FUNCTION_BLOCK FB_ESSMonitoringMCU500x
VAR_INPUT
    nEcMasterNetId: T_AmsNetId;
END_VAR
VAR_OUTPUT
    aErrorID: ARRAY [1..nMaxAlarms] OF INT;
    aErrorMsg: ARRAY [1..nMaxAlarms] OF STRING;
    nEcMasterFramesLost: UDINT;
    nCPULoad: UDINT;
    fCycleExecTime_ms: REAL;
    nAlarmGrpBitNumber: UDINT;
END_VAR
VAR
    //Outputs
    {attribute 'TcLinkTo' := 'TIID^Device 2 (EtherCAT)^Term 1 (EK1100)^Term 8 (EL2014)^DIG Outputs^Channel 1^Output'}
    bStatusLED AT %Q*: BOOL;
    {attribute 'TcLinkTo' := 'TIID^Device 2 (EtherCAT)^Term 1 (EK1100)^Term 7 (EL2014)^DIG Outputs^Channel 4^Output'}
    bAcknowledgeLED AT %Q*: BOOL;
    {attribute 'TcLinkTo' := 'TIID^Device 2 (EtherCAT)^Term 1 (EK1100)^Term 8 (EL2014)^DIG Outputs^Channel 2^Output'}
    bEStopLED AT %Q*: BOOL;
    {attribute 'TcLinkTo' := 'TIID^Device 2 (EtherCAT)^Term 1 (EK1100)^Term 8 (EL2014)^DIG Outputs^Channel 3^Output'}
    bEmergencyLED AT %Q*: BOOL;
    {attribute 'TcLinkTo' := 'TIID^Device 2 (EtherCAT)^Term 1 (EK1100)^Term 8 (EL2014)^DIG Outputs^Channel 4^Output'}
    bAbnormalLED AT %Q*: BOOL;

    //Inputs
    {attribute 'TcLinkTo' := 'TIID^Device 2 (EtherCAT)^Term 1 (EK1100)^Term 4 (EL1808)^Channel 1^Input'}
    b24VDC1_OK AT %I*: BOOL;
    {attribute 'TcLinkTo' := 'TIID^Device 2 (EtherCAT)^Term 1 (EK1100)^Term 4 (EL1808)^Channel 2^Input'}
    b24VDC2_OK AT %I*: BOOL;
    {attribute 'TcLinkTo' := 'TIID^Device 2 (EtherCAT)^Term 1 (EK1100)^Term 4 (EL1808)^Channel 3^Input'}
    b24VDC3_OK AT %I*: BOOL;
    {attribute 'TcLinkTo' := 'TIID^Device 2 (EtherCAT)^Term 1 (EK1100)^Term 4 (EL1808)^Channel 4^Input'}
    b48VDC1_OK AT %I*: BOOL;
    {attribute 'TcLinkTo' := 'TIID^Device 2 (EtherCAT)^Term 1 (EK1100)^Term 4 (EL1808)^Channel 5^Input'}
    b48VDC2_OK AT %I*: BOOL;
    {attribute 'TcLinkTo' := 'TIID^Device 2 (EtherCAT)^Term 1 (EK1100)^Term 4 (EL1808)^Channel 6^Input'}
    b48VDC3_OK AT %I*: BOOL;
    {attribute 'TcLinkTo' := 'TIID^Device 2 (EtherCAT)^Term 1 (EK1100)^Term 4 (EL1808)^Channel 7^Input'}
    b48VDC4_OK AT %I*: BOOL;
    {attribute 'TcLinkTo' := 'TIID^Device 2 (EtherCAT)^Term 1 (EK1100)^Term 3 (EL1808)^Channel 1^Input'}
    bFuse1_OK AT %I*: BOOL;
    {attribute 'TcLinkTo' := 'TIID^Device 2 (EtherCAT)^Term 1 (EK1100)^Term 3 (EL1808)^Channel 2^Input'}
    bFuse2_OK AT %I*: BOOL;
    {attribute 'TcLinkTo' := 'TIID^Device 2 (EtherCAT)^Term 1 (EK1100)^Term 3 (EL1808)^Channel 3^Input'}
    bFuse3_OK AT %I*: BOOL;
    {attribute 'TcLinkTo' := 'TIID^Device 2 (EtherCAT)^Term 1 (EK1100)^Term 3 (EL1808)^Channel 4^Input'}
    bFuse4_OK AT %I*: BOOL;
    {attribute 'TcLinkTo' := 'TIID^Device 2 (EtherCAT)^Term 1 (EK1100)^Term 3 (EL1808)^Channel 5^Input'}
    bFuse5_OK AT %I*: BOOL;
    {attribute 'TcLinkTo' := 'TIID^Device 2 (EtherCAT)^Term 1 (EK1100)^Term 3 (EL1808)^Channel 6^Input'}
    bFuse6_OK AT %I*: BOOL;
    {attribute 'TcLinkTo' := 'TIID^Device 2 (EtherCAT)^Term 1 (EK1100)^Term 3 (EL1808)^Channel 7^Input'}
    bFuse7_OK AT %I*: BOOL;
    {attribute 'TcLinkTo' := 'TIID^Device 2 (EtherCAT)^Term 1 (EK1100)^Term 3 (EL1808)^Channel 8^Input'}
    bFuse8_OK AT %I*: BOOL;
    {attribute 'TcLinkTo' := 'TIID^Device 2 (EtherCAT)^Term 1 (EK1100)^Term 5 (EL1808)^Channel 1^Input'}
    bEStop1Triggered AT %I*: BOOL;
    {attribute 'TcLinkTo' := 'TIID^Device 2 (EtherCAT)^Term 1 (EK1100)^Term 5 (EL1808)^Channel 2^Input'}
    bSTO1Triggered AT %I*: BOOL;
    {attribute 'TcLinkTo' := 'TIID^Device 2 (EtherCAT)^Term 1 (EK1100)^Term 5 (EL1808)^Channel 3^Input'}
    bEStop2Triggered AT %I*: BOOL;
    {attribute 'TcLinkTo' := 'TIID^Device 2 (EtherCAT)^Term 1 (EK1100)^Term 5 (EL1808)^Channel 4^Input'}
    bSTO2Triggered AT %I*: BOOL;
    {attribute 'TcLinkTo' := 'TIID^Device 2 (EtherCAT)^Term 1 (EK1100)^Term 6 (EL1808)^Channel 2^Input'}
    bMCB_OK AT %I*: BOOL;
    {attribute 'TcLinkTo' := 'TIID^Device 2 (EtherCAT)^Term 1 (EK1100)^Term 6 (EL1808)^Channel 3^Input'}
    bSPD_OK AT %I*: BOOL;
    {attribute 'TcLinkTo' := 'TIID^Device 2 (EtherCAT)^Term 1 (EK1100)^Term 6 (EL1808)^Channel 4^Input'}
    bDoorClosed AT %I*: BOOL;
    {attribute 'TcLinkTo' := 'TIID^Device 2 (EtherCAT)^Term 1 (EK1100)^Term 6 (EL1808)^Channel 5^Input'}
    bAcknowledgeButton AT %I*: BOOL;
    {attribute 'TcLinkTo' := 'TIID^Device 2 (EtherCAT)^Term 1 (EK1100)^Term 9 (EL3214)^RTD Inputs Channel 1^Value'}
    nTemp1 AT %I*: INT;
    {attribute 'TcLinkTo' := 'TIID^Device 2 (EtherCAT)^Term 1 (EK1100)^Term 9 (EL3214)^RTD Inputs Channel 2^Value'}
    nTemp2 AT %I*: INT;
    {attribute 'TcLinkTo' := 'TIID^Device 2 (EtherCAT)^Term 1 (EK1100)^Term 9 (EL3214)^RTD Inputs Channel 3^Value'}
    nTemp3 AT %I*: INT;
    {attribute 'TcLinkTo' := 'TIID^Device 2 (EtherCAT)^Term 1 (EK1100)^Term 9 (EL3214)^RTD Inputs Channel 4^Value'}
    nTemp4 AT %I*: INT;
    {attribute 'TcLinkTo' := 'TIID^Device 2 (EtherCAT)^Inputs^DevState'}
    nEcMasterDevState AT %I*: UINT;

    aAlarmList: ARRAY [1..nMaxAlarms] OF ST_MonitoringAlarm := [
(*[1]*)(nErrorID:=241, sErrorMsg:='The DC OK Status from PS 24V-1 is OFF.', nStatusLED:=E_MonitoringLedFunction.eFast, nAbnormalLED:=E_MonitoringLedFunction.eSteady, nEmergencyLED:=E_MonitoringLedFunction.eSteady, nAcknowledgeLED:=E_MonitoringLedFunction.eSteady),
(*[2]*)(nErrorID:=242, sErrorMsg:='The DC OK Status from PS 24V-2 is OFF.', nStatusLED:=E_MonitoringLedFunction.eFast, nAbnormalLED:=E_MonitoringLedFunction.eSteady, nEmergencyLED:=E_MonitoringLedFunction.eSteady, nAcknowledgeLED:=E_MonitoringLedFunction.eSteady),
(*[3]*)(nErrorID:=243, sErrorMsg:='The DC OK Status from PS 24V-3 is OFF.', nStatusLED:=E_MonitoringLedFunction.eFast, nAbnormalLED:=E_MonitoringLedFunction.eSteady, nEmergencyLED:=E_MonitoringLedFunction.eSteady, nAcknowledgeLED:=E_MonitoringLedFunction.eSteady),
(*[4]*)(nErrorID:=481, sErrorMsg:='The DC OK Status from PS 48V-1 is OFF.', nStatusLED:=E_MonitoringLedFunction.eFast, nAbnormalLED:=E_MonitoringLedFunction.eSteady, nEmergencyLED:=E_MonitoringLedFunction.eSteady, nAcknowledgeLED:=E_MonitoringLedFunction.eSteady),
(*[5]*)(nErrorID:=482, sErrorMsg:='The DC OK Status from PS 48V-2 is OFF.', nStatusLED:=E_MonitoringLedFunction.eFast, nAbnormalLED:=E_MonitoringLedFunction.eSteady, nEmergencyLED:=E_MonitoringLedFunction.eSteady, nAcknowledgeLED:=E_MonitoringLedFunction.eSteady),
(*[6]*)(nErrorID:=483, sErrorMsg:='The DC OK Status from PS 48V-3 is OFF.', nStatusLED:=E_MonitoringLedFunction.eFast, nAbnormalLED:=E_MonitoringLedFunction.eSteady, nEmergencyLED:=E_MonitoringLedFunction.eSteady, nAcknowledgeLED:=E_MonitoringLedFunction.eSteady),
(*[7]*)(nErrorID:=484, sErrorMsg:='The DC OK Status from PS 48V-4 is OFF.', nStatusLED:=E_MonitoringLedFunction.eFast, nAbnormalLED:=E_MonitoringLedFunction.eSteady, nEmergencyLED:=E_MonitoringLedFunction.eSteady, nAcknowledgeLED:=E_MonitoringLedFunction.eSteady),
(*[8]*)(nErrorID:=11, sErrorMsg:='MCB OK status is OFF', nStatusLED:=E_MonitoringLedFunction.eFast, nAbnormalLED:=E_MonitoringLedFunction.eSteady, nEmergencyLED:=E_MonitoringLedFunction.eSteady, nAcknowledgeLED:=E_MonitoringLedFunction.eSteady),
(*[9]*)(nErrorID:=12, sErrorMsg:='SPD OK status is OFF', nStatusLED:=E_MonitoringLedFunction.eFast, nAbnormalLED:=E_MonitoringLedFunction.eSteady, nEmergencyLED:=E_MonitoringLedFunction.eSteady, nAcknowledgeLED:=E_MonitoringLedFunction.eSteady),
(*[10]*)(nErrorID:=13, sErrorMsg:='Cabinet door Opened', nStatusLED:=E_MonitoringLedFunction.eSteady, nAbnormalLED:=E_MonitoringLedFunction.eSteady, nEmergencyLED:=E_MonitoringLedFunction.eSteady, nAcknowledgeLED:=E_MonitoringLedFunction.eUndefined),
(*[11]*)(nErrorID:=301, sErrorMsg:='Fuse 1 tripped', nStatusLED:=E_MonitoringLedFunction.eUndefined, nAbnormalLED:=E_MonitoringLedFunction.eSteady, nEmergencyLED:=E_MonitoringLedFunction.eUndefined, nAcknowledgeLED:=E_MonitoringLedFunction.eSteady),
(*[12]*)(nErrorID:=302, sErrorMsg:='Fuse 2 tripped', nStatusLED:=E_MonitoringLedFunction.eSlow, nAbnormalLED:=E_MonitoringLedFunction.eSteady, nEmergencyLED:=E_MonitoringLedFunction.eSteady, nAcknowledgeLED:=E_MonitoringLedFunction.eSteady),
(*[13]*)(nErrorID:=303, sErrorMsg:='Fuse 3 tripped', nStatusLED:=E_MonitoringLedFunction.eSlow, nAbnormalLED:=E_MonitoringLedFunction.eSteady, nEmergencyLED:=E_MonitoringLedFunction.eSteady, nAcknowledgeLED:=E_MonitoringLedFunction.eSteady),
(*[14]*)(nErrorID:=304, sErrorMsg:='Fuse 4 tripped', nStatusLED:=E_MonitoringLedFunction.eSlow, nAbnormalLED:=E_MonitoringLedFunction.eSteady, nEmergencyLED:=E_MonitoringLedFunction.eUndefined, nAcknowledgeLED:=E_MonitoringLedFunction.eSteady),
(*[15]*)(nErrorID:=305, sErrorMsg:='Fuse 5 tripped', nStatusLED:=E_MonitoringLedFunction.eSlow, nAbnormalLED:=E_MonitoringLedFunction.eSteady, nEmergencyLED:=E_MonitoringLedFunction.eUndefined, nAcknowledgeLED:=E_MonitoringLedFunction.eSteady),
(*[16]*)(nErrorID:=306, sErrorMsg:='Fuse 6 tripped', nStatusLED:=E_MonitoringLedFunction.eSlow, nAbnormalLED:=E_MonitoringLedFunction.eSteady, nEmergencyLED:=E_MonitoringLedFunction.eUndefined, nAcknowledgeLED:=E_MonitoringLedFunction.eSteady),
(*[17]*)(nErrorID:=307, sErrorMsg:='Fuse 7 tripped', nStatusLED:=E_MonitoringLedFunction.eSlow, nAbnormalLED:=E_MonitoringLedFunction.eSteady, nEmergencyLED:=E_MonitoringLedFunction.eUndefined, nAcknowledgeLED:=E_MonitoringLedFunction.eSteady),
(*[18]*)(nErrorID:=308, sErrorMsg:='Fuse 8 tripped', nStatusLED:=E_MonitoringLedFunction.eSlow, nAbnormalLED:=E_MonitoringLedFunction.eSteady, nEmergencyLED:=E_MonitoringLedFunction.eUndefined, nAcknowledgeLED:=E_MonitoringLedFunction.eSteady),
(*[19]*)(nErrorID:=501, sErrorMsg:='E-Stop 1 active', nStatusLED:=E_MonitoringLedFunction.eSteady, nAbnormalLED:=E_MonitoringLedFunction.eSteady, nEmergencyLED:=E_MonitoringLedFunction.eUndefined, nAcknowledgeLED:=E_MonitoringLedFunction.eUndefined, nEStopLED:=E_MonitoringLedFunction.eSteady),
(*[20]*)(nErrorID:=511, sErrorMsg:='STO axis 1 active', nStatusLED:=E_MonitoringLedFunction.eFast, nAbnormalLED:=E_MonitoringLedFunction.eSteady, nEmergencyLED:=E_MonitoringLedFunction.eUndefined, nAcknowledgeLED:=E_MonitoringLedFunction.eUndefined),
(*[21]*)(nErrorID:=502, sErrorMsg:='E-Stop 2 active', nStatusLED:=E_MonitoringLedFunction.eSteady, nAbnormalLED:=E_MonitoringLedFunction.eSteady, nEmergencyLED:=E_MonitoringLedFunction.eUndefined, nAcknowledgeLED:=E_MonitoringLedFunction.eUndefined, nEStopLED:=E_MonitoringLedFunction.eSteady),
(*[22]*)(nErrorID:=512, sErrorMsg:='STO axis 2 active', nStatusLED:=E_MonitoringLedFunction.eFast, nAbnormalLED:=E_MonitoringLedFunction.eSteady, nEmergencyLED:=E_MonitoringLedFunction.eUndefined, nAcknowledgeLED:=E_MonitoringLedFunction.eUndefined),
(*[23]*)(nErrorID:=14, sErrorMsg:='Temperature 1 too high', nStatusLED:=E_MonitoringLedFunction.eUndefined, nAbnormalLED:=E_MonitoringLedFunction.eSteady, nEmergencyLED:=E_MonitoringLedFunction.eSteady, nAcknowledgeLED:=E_MonitoringLedFunction.eUndefined),
(*[24]*)(nErrorID:=15, sErrorMsg:='Temperature 2 too high', nStatusLED:=E_MonitoringLedFunction.eUndefined, nAbnormalLED:=E_MonitoringLedFunction.eSteady, nEmergencyLED:=E_MonitoringLedFunction.eSteady, nAcknowledgeLED:=E_MonitoringLedFunction.eUndefined),
(*[25]*)(nErrorID:=16, sErrorMsg:='Temperature 3 too high', nStatusLED:=E_MonitoringLedFunction.eUndefined, nAbnormalLED:=E_MonitoringLedFunction.eSteady, nEmergencyLED:=E_MonitoringLedFunction.eSteady, nAcknowledgeLED:=E_MonitoringLedFunction.eUndefined),
(*[26]*)(nErrorID:=17, sErrorMsg:='Temperature 4 too high', nStatusLED:=E_MonitoringLedFunction.eUndefined, nAbnormalLED:=E_MonitoringLedFunction.eSteady, nEmergencyLED:=E_MonitoringLedFunction.eSteady, nAcknowledgeLED:=E_MonitoringLedFunction.eUndefined),
(*[27]*)(nErrorID:=101, sErrorMsg:='EtherCAT Master is not ok', nStatusLED:=E_MonitoringLedFunction.eSteady, nAbnormalLED:=E_MonitoringLedFunction.eSlow, nEmergencyLED:=E_MonitoringLedFunction.eUndefined, nAcknowledgeLED:=E_MonitoringLedFunction.eUndefined),
(*[28]*)(nErrorID:=102, sErrorMsg:='At least one EtherCAT slave is not in OP state', nStatusLED:=E_MonitoringLedFunction.eSteady, nAbnormalLED:=E_MonitoringLedFunction.eSlow, nEmergencyLED:=E_MonitoringLedFunction.eSteady, nAcknowledgeLED:=E_MonitoringLedFunction.eUndefined),
(*[29]*)(nErrorID:=103, sErrorMsg:='At least one EtherCAT slave link is faulted', nStatusLED:=E_MonitoringLedFunction.eSteady, nAbnormalLED:=E_MonitoringLedFunction.eSlow, nEmergencyLED:=E_MonitoringLedFunction.eSteady, nAcknowledgeLED:=E_MonitoringLedFunction.eUndefined),
(*[30]*)(nErrorID:=104, sErrorMsg:='Overflow in PLC cycle time', nStatusLED:=E_MonitoringLedFunction.eSteady, nAbnormalLED:=E_MonitoringLedFunction.eSlow, nEmergencyLED:=E_MonitoringLedFunction.eUndefined, nAcknowledgeLED:=E_MonitoringLedFunction.eUndefined),
(*[31]*)(nErrorID:=105, sErrorMsg:='CPU Load High', nStatusLED:=E_MonitoringLedFunction.eSteady, nAbnormalLED:=E_MonitoringLedFunction.eSlow, nEmergencyLED:=E_MonitoringLedFunction.eUndefined, nAcknowledgeLED:=E_MonitoringLedFunction.eUndefined)];

    aTempErrorID: ARRAY [1..nMaxAlarms] OF INT;
    aTempErrorMsg: ARRAY [1..nMaxAlarms] OF STRING;

    aFbErrorMessageTimer: ARRAY[1..nMaxAlarms] OF TON;
    aStartErrorMsgTimer: ARRAY[1..nMaxAlarms] OF BOOL;
    aFbErrorTrig: ARRAY[1..nMaxAlarms] OF R_TRIG;

    nLEDAlarmID: INT;
    nAlarmCnt: INT;
    nAlarmBitNumber: UDINT;

    bCPUOverloaded: BOOL;
    bEcMasterError: BOOL;
    bSlaveStateNotOP: BOOL;
    bSlaveLinkError: BOOL;
    aExtraMessage: ARRAY[1..nMaxAlarms] OF STRING := [nMaxAlarms('')];
    bCycleTimeExceeded: BOOL;
    //Cpu Monitor
    fbMonitorCPU: TC_CpuUsage;
    fbUpdateCPULoadTON: TON;
    fMaxCPULoad: USINT := 85;
    //Ethercat master device state
    bEcLinkError: BOOL;
    bEcIOlocked: BOOL;
    bEcLinkErrorRedundancyAdapter: BOOL;
    bEcMissingFrame: BOOL;
    bEcOutofSendResources: BOOL;
    bEcWatchdogTriggered: BOOL;
    bEcEthernetDriverNotFound: BOOL;
    bEcIOresetActive: BOOL;
    bEcSlaveINIT: BOOL;
    bEcSlavePreOP: BOOL;
    bEcSlaveSafeOP: BOOL;
    bEcSlaveError: BOOL;
    bEcDCnotInSync: BOOL;
    //Ehtercat slave device state
    fbUpdateEcSlaveStateTON: TON;
    fbGetEcSlaveStates: FB_EcGetAllSlaveStates;
    stSlaveState: ARRAY[0..nMaxECSlaves] OF ST_EcSlaveState;
    nActualEcSlaves: INT := 0;
    i: INT;
    //Frame statistics
    fbUpdateEcMasterFrame: TON;
    fbGetEcMasterFrames: FB_EcMasterFrameStatistic;

    nAcknowledgeLED: E_MonitoringLedFunction;
    nStatusLED: E_MonitoringLedFunction;
    nAbnormalLED: E_MonitoringLedFunction;
    nEmergencyLED: E_MonitoringLedFunction;
    fbFastBlinkOn: TON;
    fbFastBlinkOff: TON;
    bFastBlink: BOOL;
    fbSlowBlinkOn: TON;
    fbSlowBlinkOff: TON;
    bSlowBlink: BOOL;

    fbAcknowledgeButtonTrig: R_TRIG;

    fbEtherCATAlarmDelayTON: TON;
    bStartEtherCATdelayTON: BOOL := FALSE;
    bEtherCATInitialized: BOOL := FALSE;
END_VAR
VAR CONSTANT
    nMaxAlarms: INT := 50;
    nMaxECSlaves: INT := 255;
    nMaxTemp: INT := 10000;
    nSlaveStateNotOPEntry: UDINT := 28;
    nSlaveLinkErrorEntry: UDINT := 29;
END_VAR

actMonitorAlarms();
actMonitorCPU();
actMonitorEtherCAT();

ACTION actMonitorAlarms:
fbAcknowledgeButtonTrig(CLK:=bAcknowledgeButton);
mSetResetAlarmsLeds();

// Reset before loop
nAlarmCnt := 0;
nAlarmBitNumber := 0;
MEMSET(ADR(aTempErrorID), 0, SIZEOF(aTempErrorID));
MEMSET(ADR(aTempErrorMsg), 0, SIZEOF(aTempErrorMsg));
nLEDAlarmID := 0;
nEmergencyLED := 0;
nAbnormalLED := 0;
nStatusLED := 0;
nAcknowledgeLED := 0;

FOR i:=1 TO nMaxAlarms DO
    afbErrorMessageTimer[i](IN:=aStartErrorMsgTimer[i], PT:=T#60S);
    aFbErrorTrig[i](clk:=aStartErrorMsgTimer[i]);
    // Update list of active alarms
    mAlarm(stAlarmData:=aAlarmList[i]);
    // Update list of active LEDs
    mLed(stAlarmData:=aAlarmList[i]);

    IF aAlarmList[i].bAlarmActive THEN
        nAlarmCnt := nAlarmCnt + 1;
        aTempErrorID[nAlarmCnt] := aAlarmList[i].nErrorID;
        aTempErrorMsg[nAlarmCnt] := CONCAT(aAlarmList[i].sErrorMsg, aExtraMessage[i]);

        mPrintErrorMessage(
            sErrorMessage:=aTempErrorMsg[nAlarmCnt],
            nErrorID:=aAlarmList[i].nErrorID);

        // Map nErrorID to nAlarmBitnumber, which later is mapped to output variable nAlarmGrpBitNumber.
        CASE aAlarmList[i].nErrorID OF
            1,4:
            nAlarmBitNumber.0 := TRUE;
            9,12,13:
            nAlarmBitNumber.1 := TRUE;
            10,11:
            nAlarmBitNumber.2 := TRUE;
            14,15:
            nAlarmBitNumber.3 := TRUE;
            21,22:
            nAlarmBitNumber.4 := TRUE;
            23,24:
            nAlarmBitNumber.5 := TRUE;
            104,105:
            nAlarmBitNumber.6 := TRUE;
            103:
            nAlarmBitNumber.7 := TRUE;
            102:
            nAlarmBitNumber.8 := TRUE;
            30:
            nAlarmBitNumber.9 := TRUE;
        END_CASE
    END_IF

    // Set the alarm LEDs according to first occurrence
    IF nLEDAlarmID = 0 AND aALarmList[i].bLedActive THEN
        nLEDAlarmID := i;
        nEmergencyLED := aAlarmList[i].nEmergencyLED;
        nAbnormalLED := aAlarmList[i].nAbnormalLED;
        nStatusLED := aAlarmList[i].nStatusLED;
        nAcknowledgeLED := aAlarmList[i].nAcknowledgeLED;
    END_IF
END_FOR


// Copy to output variables
aErrorID := aTempErrorID;
aErrorMsg := aTempErrorMsg;
nAlarmGrpBitNumber := nAlarmBitNumber;

// Handle LED blinking
fbFastBlinkOn(IN:=NOT fbFastBlinkOff.q , PT:=T#250MS , Q=> , ET=> );
fbFastBlinkOff(IN:=fbFastBlinkOn.Q , PT:=T#250MS , Q=> , ET=> );
bFastBlink := fbFastBlinkOn.q;

fbSlowBlinkOn(IN:=NOT fbSlowBlinkOff.q , PT:=T#750MS , Q=> , ET=> );
fbSlowBlinkOff(IN:=fbSlowBlinkOn.Q , PT:=T#750MS , Q=> , ET=> );
bSlowBlink := fbSlowBlinkOn.q;

bEmergencyLED :=
    (nEmergencyLED = E_MonitoringLedFunction.eSteady)
    OR (nEmergencyLED = E_MonitoringLedFunction.eFast AND bFastBlink)
    OR (nEmergencyLED = E_MonitoringLedFunction.eSlow AND bSlowBlink);
bAbnormalLED :=
    (nAbnormalLED = E_MonitoringLedFunction.eSteady)
    OR (nAbnormalLED = E_MonitoringLedFunction.eFast AND bFastBlink)
    OR (nAbnormalLED = E_MonitoringLedFunction.eSlow AND bSlowBlink);
bStatusLED :=
    (nStatusLED = E_MonitoringLedFunction.eSteady)
    OR (nStatusLED = E_MonitoringLedFunction.eFast AND bFastBlink)
    OR (nStatusLED = E_MonitoringLedFunction.eSlow AND bSlowBlink);
bAcknowledgeLED :=
    (nAcknowledgeLED = E_MonitoringLedFunction.eSteady)
    OR (nAcknowledgeLED = E_MonitoringLedFunction.eFast AND bFastBlink)
    OR (nAcknowledgeLED = E_MonitoringLedFunction.eSlow AND bSlowBlink);
END_ACTION

ACTION actMonitorCPU:
//Cpu Monitor
fbUpdateCPULoadTON(IN:=NOT fbUpdateCPULoadTON.q , PT:=T#100MS , Q=> , ET=> );
fbMonitorCPU(START:=fbUpdateCPULoadTON.q, TMOUT:= T#5S);

bCPUOverloaded := fbMonitorCPU.USAGE > fMaxCPULoad;
nCPULoad := fbMonitorCPU.USAGE;

fCycleExecTime_ms := UDINT_TO_REAL(_TaskInfo[fbGetCurTaskIndex.index].LastExecTime) / 10000;
bCycleTimeExceeded := _TaskInfo[fbGetCurTaskIndex.index].CycleTimeExceeded;
END_ACTION

ACTION actMonitorEtherCAT:
//Read frames
fbUpdateEcMasterFrame(IN:=NOT fbUpdateEcMasterFrame.q , PT:=T#1000MS , Q=> , ET=> );
fbGetEcMasterFrames(sNetId:= nEcMasterNetId, bExecute:= fbUpdateEcMasterFrame.q);

nEcMasterFramesLost := fbGetEcMasterFrames.nLostFrames;


//Check ethercat slave device state
fbUpdateEcSlaveStateTON(IN:=NOT fbUpdateEcSlaveStateTON.q , PT:=T#100MS , Q=> , ET=> );
fbGetEcSlaveStates(
    sNetId:=nEcMasterNetId,
    pStateBuf:=ADR(stSlaveState),
    cbBufLen:=SIZEOF(stSlaveState),
    bExecute:=fbUpdateEcSlaveStateTON.q);
nActualEcSlaves:=UINT_TO_INT(fbGetEcSlaveStates.nSlaves);

fbEtherCATAlarmDelayTON(IN:=bStartEtherCATdelayTON, PT:=T#1S);

IF fbEtherCATAlarmDelayTON.Q THEN
    bStartEtherCATdelayTON := FALSE;
    bEtherCATInitialized := TRUE;
END_IF

IF bEtherCATInitialized THEN
    FOR i:=0 TO nActualEcSlaves-1 DO
        IF i = 0 THEN
            bSlaveStateNotOP := FALSE;
            bSlaveLinkError := FALSE;
            aExtraMessage[nSlaveStateNotOPEntry] := ', Slave Nbr: ';
            aExtraMessage[nSlaveLinkErrorEntry] := ', Slave Nbr: ';
        END_IF

        IF stSlaveState[i].deviceState <> EC_DEVICE_STATE_OP THEN
            bSlaveStateNotOP := TRUE;
            CONCAT(STR1:=aExtraMessage[nSlaveStateNotOPEntry], STR2:=INT_TO_STRING(i));
            CONCAT(STR1:=aExtraMessage[nSlaveStateNotOPEntry], STR2:=', ');
        END_IF

        IF stSlaveState[i].linkState <> EC_LINK_STATE_OK  THEN
            bSlaveLinkError := TRUE;
            CONCAT(STR1:=aExtraMessage[nSlaveLinkErrorEntry], STR2:=INT_TO_STRING(i));
            CONCAT(STR1:=aExtraMessage[nSlaveLinkErrorEntry], STR2:=', ');
        END_IF
    END_FOR
ELSE
    bStartEtherCATdelayTON := TRUE;
END_IF

//Check ethercat master device state
bEcLinkError := nEcMasterDevState.0;
bEcIOlocked := nEcMasterDevState.1;
bEcLinkErrorRedundancyAdapter := nEcMasterDevState.2;
bEcMissingFrame := nEcMasterDevState.3;
bEcOutofSendResources := nEcMasterDevState.4;
bEcWatchdogTriggered := nEcMasterDevState.5;
bEcEthernetDriverNotFound := nEcMasterDevState.6;
bEcIOresetActive := nEcMasterDevState.7;
bEcSlaveINIT := nEcMasterDevState.8;
bEcSlavePreOP := nEcMasterDevState.9;
bEcSlaveSafeOP := nEcMasterDevState.10;
bEcSlaveError := nEcMasterDevState.11;
bEcDCnotInSync := nEcMasterDevState.12;

bEcMasterError := nEcMasterDevState > 0;
END_ACTION

METHOD mAlarm : BOOL
VAR_IN_OUT
    stAlarmData: ST_MonitoringAlarm;
END_VAR
IF stAlarmData.bAlarmSet THEN
    stAlarmData.bAlarmActive := TRUE;
ELSIF stAlarmData.bAlarmReset THEN
    stAlarmData.bAlarmActive := FALSE;
END_IF
END_METHOD

METHOD mLed : BOOL
VAR_IN_OUT
    stAlarmData: ST_MonitoringAlarm;
END_VAR
IF stAlarmData.bLedSet THEN
    stAlarmData.bLedActive := TRUE;
ELSIF stAlarmData.bLedReset THEN
    stAlarmData.bLedActive := FALSE;
END_IF
END_METHOD

METHOD mPrintErrorMessage : BOOL
VAR_INPUT
    sErrorMessage: STRING;
    nErrorID: INT;
END_VAR
VAR
    sFullErrorMessage: STRING;
END_VAR
sFullErrorMessage := CONCAT(STR1:='ERROR. ErrorID: ', STR2:=INT_TO_STRING(nErrorID));
sFullErrorMessage := CONCAT(STR1:=sFullErrorMessage, STR2:='. ');
sFullErrorMessage := CONCAT(STR1:=sFullErrorMessage, STR2:=sErrorMessage);

IF aAlarmList[i].bAlarmActive THEN
    aStartErrorMsgTimer[i]:=TRUE;
    IF afbErrorTrig[i].Q THEN
        ADSLOGSTR(
            msgCtrlMask:=ADSLOG_MSGTYPE_ERROR,
            msgFmtStr:='%s',
            strArg:=sFullErrorMessage);
    END_IF

    IF aFbErrorMessageTimer[i].Q THEN
        aStartErrorMsgTimer[i]:=FALSE;
    END_IF
END_IF
END_METHOD

METHOD mSetResetAlarmsLeds : BOOL
VAR_INST
    index: INT;
END_VAR
IF NOT b24VDC1_OK THEN
    aAlarmList[1].bAlarmSet := TRUE;
    aAlarmList[1].bAlarmReset := FALSE;
END_IF

IF NOT b24VDC2_OK THEN
    aAlarmList[2].bAlarmSet := TRUE;
    aAlarmList[2].bAlarmReset := FALSE;
END_IF

IF NOT b24VDC3_OK THEN
    aAlarmList[3].bAlarmSet := TRUE;
    aAlarmList[3].bAlarmReset := FALSE;
END_IF

IF NOT b48VDC1_OK THEN
    aAlarmList[4].bAlarmSet := TRUE;
    aAlarmList[4].bAlarmReset := FALSE;
END_IF

IF NOT b48VDC2_OK THEN
    aAlarmList[5].bAlarmSet := TRUE;
    aAlarmList[5].bAlarmReset := FALSE;
END_IF

IF NOT b48VDC3_OK THEN
    aAlarmList[6].bAlarmSet := TRUE;
    aAlarmList[6].bAlarmReset := FALSE;
END_IF

IF NOT b48VDC4_OK THEN
    aAlarmList[7].bAlarmSet := TRUE;
    aAlarmList[7].bAlarmReset := FALSE;
END_IF

IF NOT bMCB_OK THEN
    aAlarmList[8].bAlarmSet := TRUE;
    aAlarmList[8].bAlarmReset := FALSE;
END_IF

IF NOT bSPD_OK THEN
    aAlarmList[9].bAlarmSet := TRUE;
    aAlarmList[9].bAlarmReset := FALSE;
END_IF

IF NOT bDoorClosed THEN
    aAlarmList[10].bAlarmSet := TRUE;
    aAlarmList[10].bAlarmReset := FALSE;
ELSE
    aAlarmList[10].bAlarmSet := FALSE;
    aAlarmList[10].bAlarmReset:= TRUE;
END_IF

IF NOT bFuse1_OK THEN
    aAlarmList[11].bAlarmSet := TRUE;
    aAlarmList[11].bAlarmReset := FALSE;
END_IF

IF bFuse2_OK THEN
    aAlarmList[12].bAlarmSet := TRUE;
    aAlarmList[12].bAlarmReset := FALSE;
END_IF

IF bFuse3_OK THEN
    aAlarmList[13].bAlarmSet := TRUE;
    aAlarmList[13].bAlarmReset := FALSE;
END_IF

IF NOT bFuse4_OK THEN
    aAlarmList[14].bAlarmSet := TRUE;
    aAlarmList[14].bAlarmReset := FALSE;
END_IF

IF NOT bFuse5_OK THEN
    aAlarmList[15].bAlarmSet := TRUE;
    aAlarmList[15].bAlarmReset := FALSE;
END_IF

IF NOT bFuse6_OK THEN
    aAlarmList[16].bAlarmSet := TRUE;
    aAlarmList[16].bAlarmReset := FALSE;
END_IF

IF NOT bFuse7_OK THEN
    aAlarmList[17].bAlarmSet := TRUE;
    aAlarmList[17].bAlarmReset := FALSE;
END_IF

IF NOT bFuse8_OK THEN
    aAlarmList[18].bAlarmSet := TRUE;
    aAlarmList[18].bAlarmReset := FALSE;
END_IF

IF NOT bEStop1Triggered THEN
    aAlarmList[19].bAlarmSet := TRUE;
    aAlarmList[19].bAlarmReset := FALSE;
ELSE
    aAlarmList[19].bAlarmSet := FALSE;
    aAlarmList[19].bAlarmReset:= TRUE;
END_IF

IF NOT bSTO1Triggered THEN
    aAlarmList[20].bAlarmSet := TRUE;
    aAlarmList[20].bAlarmReset := FALSE;
ELSE
    aAlarmList[20].bAlarmSet := FALSE;
    aAlarmList[20].bAlarmReset:= TRUE;
END_IF

IF NOT bEStop2Triggered THEN
    aAlarmList[21].bAlarmSet := TRUE;
    aAlarmList[21].bAlarmReset := FALSE;
ELSE
    aAlarmList[21].bAlarmSet := FALSE;
    aAlarmList[21].bAlarmReset:= TRUE;
END_IF

IF NOT bSTO2Triggered THEN
    aAlarmList[22].bAlarmSet := TRUE;
    aAlarmList[22].bAlarmReset := FALSE;
ELSE
    aAlarmList[22].bAlarmSet := FALSE;
    aAlarmList[22].bAlarmReset:= TRUE;
END_IF

IF nTemp1 > nMaxTemp THEN
    aAlarmList[23].bAlarmSet := TRUE;
    aAlarmList[23].bAlarmReset := FALSE;
ELSE
    aAlarmList[23].bAlarmSet := FALSE;
    aAlarmList[23].bAlarmReset:= TRUE;
END_IF

IF nTemp2 > nMaxTemp THEN
    aAlarmList[24].bAlarmSet := TRUE;
    aAlarmList[24].bAlarmReset := FALSE;
ELSE
    aAlarmList[24].bAlarmSet := FALSE;
    aAlarmList[24].bAlarmReset:= TRUE;
END_IF

IF nTemp3 > nMaxTemp THEN
    aAlarmList[25].bAlarmSet := TRUE;
    aAlarmList[25].bAlarmReset := FALSE;
ELSE
    aAlarmList[25].bAlarmSet := FALSE;
    aAlarmList[25].bAlarmReset:= TRUE;
END_IF

IF nTemp4 > nMaxTemp THEN
    aAlarmList[26].bAlarmSet := TRUE;
    aAlarmList[26].bAlarmReset := FALSE;
ELSE
    aAlarmList[26].bAlarmSet := FALSE;
    aAlarmList[26].bAlarmReset:= TRUE;
END_IF

IF bEcMasterError THEN
    aAlarmList[27].bAlarmSet := TRUE;
    aAlarmList[27].bAlarmReset := FALSE;
ELSE
    aAlarmList[27].bAlarmSet := FALSE;
    aAlarmList[27].bAlarmReset:= TRUE;
END_IF

IF bSlaveStateNotOP THEN
    aAlarmList[28].bAlarmSet := TRUE;
    aAlarmList[28].bAlarmReset := FALSE;
ELSE
    aAlarmList[28].bAlarmSet := FALSE;
    aAlarmList[28].bAlarmReset:= TRUE;
END_IF

IF bSlaveLinkError THEN
    aAlarmList[29].bAlarmSet := TRUE;
    aAlarmList[29].bAlarmReset := FALSE;
ELSE
    aAlarmList[29].bAlarmSet := FALSE;
    aAlarmList[29].bAlarmReset:= TRUE;
END_IF

IF bCycleTimeExceeded THEN
    aAlarmList[30].bAlarmSet := TRUE;
    aAlarmList[30].bAlarmReset := FALSE;
ELSE
    aAlarmList[30].bAlarmSet := FALSE;
    aAlarmList[30].bAlarmReset:= TRUE;
END_IF

IF bCPUOverloaded THEN
    aAlarmList[31].bAlarmSet := TRUE;
    aAlarmList[31].bAlarmReset := FALSE;
ELSE
    aAlarmList[31].bAlarmSet := FALSE;
    aAlarmList[31].bAlarmReset:= TRUE;
END_IF

//Reset selected alarms just when acknowledge button has been pressed
IF fbAcknowledgeButtonTrig.Q THEN
    FOR index:=1 TO 18 DO //just until 18, the rest should be reset when they dissappear, no need for acknowledge
        IF index <> 10 THEN //eStop and STO will be reset automatically via HW
            aAlarmList[index].bAlarmSet := FALSE;
            aAlarmList[index].bAlarmReset := TRUE;
        END_IF
    END_FOR
END_IF
END_METHOD

END_FUNCTION_BLOCK

(* stored: Version 1.1.0.1
   POU FB_ESSMonitoringMCU500x: Id {dc25224c-2805-4e0c-98fe-daa6f852a4e2}, SpecialFunc None
   Action actMonitorAlarms: Id {05cd06da-6727-4135-9b29-65a4335223b8}
   Action actMonitorCPU: Id {db0cbd89-0ab0-45d1-9643-6542a9f72fa2}
   Action actMonitorEtherCAT: Id {a4594d19-0db5-4810-8e12-099bc24ca287}
   Method mAlarm: Id {bc357e09-9ee8-4234-8c76-7cdeb0e72989}
   Method mLed: Id {e7c0d21c-5d75-0ad9-14e4-781003dce579}
   Method mPrintErrorMessage: Id {3e321397-22af-4d7e-a9bd-c132b0a3b842}
   Method mSetResetAlarmsLeds: Id {1241012c-ae73-450a-94a3-e603ad15f437} *)
